// TIA Portal V20 export
TYPE "sAxis_Status"
   STRUCT
      bAxisReady : Bool;   // 轴通讯正常
      bAxisEnabled : Bool;   // 轴使能
      bjogForward : Bool;   // 轴正点中
      bjogBackward : Bool;   // 轴反点中
      bHomed : Bool;   // 轴归零完成
      bAtHome : Bool;   // 轴在零位
      bSstill : Bool;   // 轴静止
      bAxisBusy : Bool;   // 轴运行中
      bAxisSyned : Bool;   // 同步上
      bAxisError : Bool;   // 轴报警
      bAtPos : Array[0..15] of Bool;   // Ausgang Aufwärts / 在目标位置上
      bPosDone : Array[0..15] of Bool;   // 定位完成
      bPosing : Array[0..15] of Bool;   // Ausgang Aufwärts / 定位中
      bRelPosDone : Bool;   // 相对定位完成
      rActPos : LReal;   // 实际位置
      rActSpeed : LReal;   // 实际速度
      iAxisFaultNum : UDInt;   // 轴报警代码
      iDriveFaultNum : UDInt;   // 驱动报警代码
      iFBStatus : Word;   // 运动功能块状态
      iMCStatus : Word;   // 运动指令状态
      rDriveTorque : LReal;   // 驱动扭矩
      rDriveTemp : LReal;   // 驱动温度
      rDriveRpm : LReal;   // 驱动转速
      wAxisName : WString[24] := WSTRING#'No axis';   // Name of axis
      mybool : Array[0..5] of Bool;   // 备用
      myLreal : Array[0..5] of LReal;   // 备用
   END_STRUCT;
END_TYPE
